(* IEC 61131-3 sources: std_i2980_v2.06_cp053/Source/IMM/ieccontrol/PDP1 (part 3) *)

(* ---- ABRecorderPQ.pu ---- *)
(*
@h    ! WARNING !
@h    The Kemro K2 system (including software) only meets category B according to EN 954-1,
@h    thus it is not intended for usage in safety-relevant control applications in the field
@h    of personal safety (e.g. emergency stop).
@h    To implement potentially necessary safety-relevant control tasks, always use additional
@h    external safety devices that are intended for the particular purpose, and meet the necessary
@h    functional safety.
@h    For further information see EN 954-1 (EN ISO 13849-1) and/or the K2-x00 user manual, chapter
@h    "CE conformity, directives and standards".

*)

IMPORT_OVER_LISTFILE
 START_PROCESS_ALGORITHM
, STOP_PROCESS_ALGORITHM
, GET_SYNC_REFTO
, cCompMold
, tyMovementTrigger
, tevMovementState
, tnOperationMode
, KMB_MeasureBlock2
, KMB_Status
, KMB_CurveResult
, KMB_Curve
, KMB_CreateProfileData
, KSYS_Status
, tevMovementStateData
, KMB_ProfileInfo

END_IMPORT

ALGORITHM_BLOCK ABRecorderPQ #DUMMY_EDIT_BLOCK

SYSTEM_VAR
 sv_TriggerIdxRecPQ : UDINT;
 sv_OperationMode : tnOperationMode ;
 sv_bPQChartHoldRun : BOOL (* PQ chart hold / run *);
END_VAR

SYSTEM_OBJECT
 TaskVis : TASK;
 TaskInject : TASK;
 evMovementState : tevMovementState;
END_OBJECT

VAR
 myMovementTrigger : tyMovementTrigger;
 mevStart : tevMovementState;
 mpbPumpDeviceReady : REFTO BOOL;
 abMeasure : KMB_MeasureBlock2;
 mpiTriggerIdx : REFTO UDINT;
END_VAR

FUNCTION fStartInit : BOOL
 #DUMMY_EDIT_BLOCK
#BEGIN_EDIT_BLOCK
(**************************************** WARNING ********************************************
 *** The KEBA Kemro K2 System including software is not intended for safety control tasks! ***
 ***                       For further information see Comment tab!                        ***
 *********************************************************************************************)

fStartInit := FALSE; //suppress warning about unused formal parameter
START_PROCESS_ALGORITHM(paInit);

;#END_EDIT_BLOCK END_FUNCTION

PROCESS_ALGORITHM paInit ON TaskVis

VAR
 status : KMB_Status;
 curveStatus : KMB_CurveResult;
 curve : KMB_Curve;
 bCreated : BOOL;
 profileData : KMB_CreateProfileData := (ProfileName:='ChartPQ',Type:=KMB_ProfileKind_PDSC,ElementCount:=10000,DataPath:='/protocol/datalogger/',CfgPath:='/workspace/data/ms_config/',ThreadPriority:=6);
 s : KSYS_Status;
END_VAR
#BEGIN_EDIT_BLOCK
(**************************************** WARNING ********************************************
 *** The KEBA Kemro K2 System including software is not intended for safety control tasks! ***
 ***                       For further information see Comment tab!                        ***
 *********************************************************************************************)

// create and init profile 'ChartPQ' of type Mic / 10000  elements
IF (NOT bCreated) THEN
   // create and configure profile for 4 ms cyclic measure
   status := abMeasure.CreateProfile(profileData);
   status := abMeasure.DisableProfileFlashPersistence();
   status := abMeasure.DisableAutoSaveConfig();
   status := abMeasure.SetMeasureTime(T#4ms);
   bCreated := TRUE;
END_IF;

(* add variables 0 .. 3: movement states *)
curve.VariableY := "Mold1.sv_bCloseActive";
curveStatus := abMeasure.AddCurve(curve);

IF (curveStatus.Status = KMB_Status_Not_Connected) THEN
   // see iec library doc and CR_0053873 "KMB_MeasureBlock2: curve is added twice"
   // if a profile has been created it will be installed async. to the IEC task
   // so it may happen that installation of profile has not been finished.
   // we have to repeat here until Status different to "not connected"
   RETURN;
END_IF;

curve.VariableY := "Mold1.sv_bOpenActive";
curveStatus := abMeasure.AddCurve(curve);

curve.VariableY := "Injection1.sv_bPlastActive";
curveStatus := abMeasure.AddCurve(curve);

curve.VariableY := "Injection1.sv_bInjectionActive";
curveStatus := abMeasure.AddCurve(curve);

(* add variables 4 .. 7: PQ set / act master *)
curve.VariableY := "Pump1.sv_KHW_ServoMaster_setValue.rVeloc";
curveStatus := abMeasure.AddCurve(curve);

curve.VariableY := "Pump1.sv_KHW_ServoMaster_actValue.rVeloc";
curveStatus := abMeasure.AddCurve(curve);

curve.VariableY := "Pump1.sv_KHW_ServoMaster_setValue.rAux[1]";
curveStatus := abMeasure.AddCurve(curve);

curve.VariableY := "Pump1.sv_KHW_ServoMaster_actValue.rAux[1]";
curveStatus := abMeasure.AddCurve(curve);

(* add optional variable 8: Q set slave 1 *)
curve.VariableY := "Pump1.sv_KHW_ServoSlave1_actValue.rVeloc";
curveStatus := abMeasure.AddCurve(curve);

(* add optional variable 9: Q set slave 2 *)
curve.VariableY := "Pump1.sv_KHW_ServoSlave2_actValue.rVeloc";
curveStatus := abMeasure.AddCurve(curve);

//////////////////////////////////////////////////////////

// init trigger variables
mpbPumpDeviceReady := GET_SYNC_REFTO("Pump1.sv_bDeviceReady", t#0s, s);
mpiTriggerIdx := @sv_TriggerIdxRecPQ;

//desciption of device and movement id

// mold fwd
myMovementTrigger[1].DeviceId.CompId := cCompMold;
myMovementTrigger[1].DeviceId.IndexId := 1;
myMovementTrigger[1].MoveId := cMoveFwd;
myMovementTrigger[1].MoveDir := cMoveFwd;

// mold bwd
myMovementTrigger[2].DeviceId.CompId := cCompMold;
myMovementTrigger[2].DeviceId.IndexId := 1;
myMovementTrigger[2].MoveId := cMoveBwd;
myMovementTrigger[2].MoveDir := cMoveBwd;

// Inject
myMovementTrigger[3].DeviceId.CompId := cCompInjection;
myMovementTrigger[3].DeviceId.IndexId := 1;
myMovementTrigger[3].MoveId := cMoveInject;
myMovementTrigger[3].MoveDir := cMoveFwd;

// Plast
myMovementTrigger[4].DeviceId.CompId := cCompInjection;
myMovementTrigger[4].DeviceId.IndexId := 1;
myMovementTrigger[4].MoveId := cMovePlast;
myMovementTrigger[4].MoveDir := cMoveBwd;

STOP_PROCESS_ALGORITHM();

;#END_EDIT_BLOCK END_ALGORITHM

EVENT_ALGORITHM evaMovementStart ON TaskInject WITH mevStart

VAR_INPUT
 evMovementStateData : tevMovementStateData;
END_VAR

VAR
 status : KMB_Status;
END_VAR
#BEGIN_EDIT_BLOCK
(**************************************** WARNING ********************************************
 *** The KEBA Kemro K2 System including software is not intended for safety control tasks! ***
 ***                       For further information see Comment tab!                        ***
 *********************************************************************************************)

//Check if in full/half automatic mode
IF sv_OperationMode < nHalfAutomatic THEN
    RETURN;
END_IF;

//Check the movement with the selection on the HMI and the Hold/Run state
//1).Mold close
//2).Mold open
//3).Inject
//4).Plast
IF (evMovementStateData.State = nActive) AND
    ((evMovementStateData.DeviceId = myMovementTrigger[sv_TriggerIdxRecPQ].DeviceId            //movement 1)-> 4)
    AND evMovementStateData.MoveId = myMovementTrigger[sv_TriggerIdxRecPQ].MoveId
    AND evMovementStateData.MoveDir = myMovementTrigger[sv_TriggerIdxRecPQ].MoveDir) OR        //mold close interposition
    (sv_TriggerIdxRecPQ = 1 AND evMovementStateData.DeviceId.CompId = cCompMold AND
     evMovementStateData.DeviceId.IndexId =1 AND evMovementStateData.MoveId = cMoveFwdInterPos AND
     evMovementStateData.MoveDir = cMoveFwd) OR                                           //mold open interposition
    (sv_TriggerIdxRecPQ = 2 AND evMovementStateData.DeviceId.CompId = cCompMold AND
     evMovementStateData.DeviceId.IndexId =1 AND evMovementStateData.MoveId = cMoveBwdInterPos AND
     evMovementStateData.MoveDir = cMoveBwd)) AND (NOT sv_bPQChartHoldRun) THEN

    // start measure
    status := abMeasure.StartMeasure(0);
END_IF;

;#END_EDIT_BLOCK END_ALGORITHM

POSTUPDATE_ALGORITHM pActivateAutoMode ON TaskVis WITH mpiTriggerIdx^

VAR
 status : KMB_Status;
END_VAR
#BEGIN_EDIT_BLOCK
(**************************************** WARNING ********************************************
 *** The KEBA Kemro K2 System including software is not intended for safety control tasks! ***
 ***                       For further information see Comment tab!                        ***
 *********************************************************************************************)

//check if trigger is selected
IF (sv_TriggerIdxRecPQ = 0) THEN
    mevStart := EMPTY;
ELSE
    status := abMeasure.StopMeasure();
    mevStart := evMovementState;
END_IF;

;#END_EDIT_BLOCK END_ALGORITHM

POSTUPDATE_ALGORITHM pActivateManualMode ON TaskInject WITH mpbPumpDeviceReady^

VAR
 status : KMB_Status;
 profileInfo : KMB_ProfileInfo;
END_VAR
#BEGIN_EDIT_BLOCK
(**************************************** WARNING ********************************************
 *** The KEBA Kemro K2 System including software is not intended for safety control tasks! ***
 ***                       For further information see Comment tab!                        ***
 *********************************************************************************************)

// trigger for manual/setup mode ... any movement
IF (sv_OperationMode <= nManual) THEN
    //Check the pump output and Hold/Run function
    IF (NOT mpbPumpDeviceReady^) AND (NOT sv_bPQChartHoldRun)THEN
         profileInfo := abMeasure.GetProfileInfo();
         // if measure still active just keep running ...
         IF (profileInfo.MeasureState = KMB_MeasureState_Inactive) THEN
            status := abMeasure.StartMeasure(0);
         END_IF;
    END_IF;
END_IF;

;#END_EDIT_BLOCK END_ALGORITHM

END_ALGORITHM_BLOCK

#END_OF_IEC_PART

@Puma @IecEditor 6 131 @Pou 25
@@@BEG_Comment@@@
@h    ! WARNING !
@h    The Kemro K2 system (including software) only meets category B according to EN 954-1,
@h    thus it is not intended for usage in safety-relevant control applications in the field
@h    of personal safety (e.g. emergency stop).
@h    To implement potentially necessary safety-relevant control tasks, always use additional
@h    external safety devices that are intended for the particular purpose, and meet the necessary
@h    functional safety.
@h    For further information see EN 954-1 (EN ISO 13849-1) and/or the K2-x00 user manual, chapter
@h    "CE conformity, directives and standards".

@@@END_Comment@@@

@BEG_Contents

@BEG_Func
@RT(17)FuncTreeContainer
3
@Var @RT(23)START_PROCESS_ALGORITHM @RT(0) @T @T @DERIVED 0 @F @RT(23)KEBA_STANDARD_PROCEDURE @F
@T
@BEG_Attrib
0 @RT(0) @RT(0)
@END_Attrib
1 1 @F @F @F @F

@Var @RT(22)STOP_PROCESS_ALGORITHM @RT(0) @T @T @DERIVED 0 @F @RT(23)KEBA_STANDARD_PROCEDURE @F
@T
@BEG_Attrib
0 @RT(0) @RT(0)
@END_Attrib
1 1 @F @F @F @F

@Var @RT(14)GET_SYNC_REFTO @RT(0) @T @T @DERIVED 0 @F @RT(22)KEBA_STANDARD_FUNCTION @F
@T
@BEG_Attrib
0 @RT(0) @RT(0)
@END_Attrib
1 1 @F @F @F @F

@END_Func

@BEG_Const
@RT(18)ConstTreeContainer
1
@Var @RT(9)cCompMold @RT(0) @T @F @DT @RT(4)DINT @RT(0) @T @T @BASIC 0 @F
@F @F
@T
@BEG_Attrib
0 @RT(3)101 @RT(14)Component Mold
@END_Attrib
1 1 @F @F @F @F

@END_Const

@BEG_Export

@BEG_Kind
@ALGORITHM_BLOCK @RT(12)ABRecorderPQ @STRUCTURED_TEXT
@RT(0) @RT(0) @RT(0)
@END_Kind

@BEG_Dcl
@RT(16)DclTreeContainer
11
@Var @RT(7)TaskVis @RT(0) @T @T @RENAMED 0 @T @T @DT @RT(4)TASK @RT(0) @T @T @BASIC 0 @F
@F @F
@T
@BEG_Attrib
3 @RT(0) @RT(0) @RT(0)
@END_Attrib
1 7 @F @F @F @F

@Var @RT(10)TaskInject @RT(0) @T @T @RENAMED 0 @T @T @DT @RT(4)TASK @RT(0) @T @T @BASIC 0 @F
@F @F
@T
@BEG_Attrib
3 @RT(0) @RT(0) @RT(0)
@END_Attrib
1 7 @F @F @F @F

@Var @RT(17)myMovementTrigger @RT(0) @T @T @DERIVED 0 @T @T @DT @RT(17)tyMovementTrigger @RT(0) @T @T @UNKNOWN 0 @F
@F @F
@T
@BEG_Attrib
3 @RT(0) @RT(0) @RT(0)
@END_Attrib
1 0 @F @F @F @F

@Var @RT(15)evMovementState @RT(0) @T @T @DERIVED 0 @T @T @DT @RT(16)tevMovementState @RT(0) @T @T @UNKNOWN 0 @F
@F @F
@T
@BEG_Attrib
3 @RT(0) @RT(0) @RT(0)
@END_Attrib
1 7 @F @F @F @F

@Var @RT(18)sv_TriggerIdxRecPQ @RT(0) @T @F @DT @RT(5)UDINT @RT(0) @T @T @BASIC 0 @F
@F @F
@T
@BEG_Attrib
3 @RT(0) @RT(0) @RT(0)
@END_Attrib
1 8 @F @F @F @F

@Var @RT(16)sv_OperationMode @RT(0) @T @T @DERIVED 0 @T @T @DT @RT(16)tnOperationMode  @RT(0) @T @T @UNKNOWN 0 @F
@F @F
@T
@BEG_Attrib
3 @RT(0) @RT(0) @RT(0)
@END_Attrib
1 8 @F @F @F @F

@Var @RT(18)sv_bPQChartHoldRun @RT(0) @T @F @DT @RT(4)BOOL @RT(0) @T @T @BASIC 0 @F
@F @F
@T
@BEG_Attrib
3 @RT(0) @RT(19)PQ chart hold / run @RT(0)
@END_Attrib
1 8 @F @F @F @F

@Var @RT(8)mevStart @RT(0) @T @T @DERIVED 0 @T @T @DT @RT(16)tevMovementState @RT(0) @T @T @UNKNOWN 0 @F
@F @F
@T
@BEG_Attrib
3 @RT(0) @RT(0) @RT(0)
@END_Attrib
1 0 @F @F @F @F

@Var @RT(18)mpbPumpDeviceReady @RT(0) @T @T @REFTO 0 @T @DT @RT(4)BOOL @RT(0) @T @T @BASIC 0 @F
@F @F
@T
@BEG_Attrib
3 @RT(0) @RT(0) @RT(0)
@END_Attrib
1 0 @F @F @F @F

@Var @RT(9)abMeasure @RT(0) @T @T @DERIVED 0 @T @T @DT @RT(17)KMB_MeasureBlock2 @RT(0) @T @T @UNKNOWN 0 @F
@F @F
@T
@BEG_Attrib
3 @RT(0) @RT(0) @RT(0)
@END_Attrib
1 0 @F @F @F @F

@Var @RT(13)mpiTriggerIdx @RT(0) @T @T @REFTO 0 @T @DT @RT(5)UDINT @RT(0) @T @T @BASIC 0 @F
@F @F
@T
@BEG_Attrib
3 @RT(0) @RT(0) @RT(0)
@END_Attrib
1 0 @F @F @F @F

@END_Dcl

@END_Export

@BEG_Body

5

@BEG_Export

@BEG_Algo
@FUNCTION @RT(10)fStartInit @STRUCTURED_TEXT
@RT(4)BOOL @RT(0) @RT(0) @F @F
@END_Algo

@BEG_Dcl
@RT(16)DclTreeContainer
0
@END_Dcl

@END_Export

@BEG_Export

@BEG_Algo
@PROCESS_ALGORITHM @RT(6)paInit @STRUCTURED_TEXT
@RT(0) @RT(0) @RT(7)TaskVis @F @F
@END_Algo

@BEG_Dcl
@RT(16)DclTreeContainer
6
@Var @RT(6)status @RT(0) @T @T @DERIVED 0 @T @T @DT @RT(10)KMB_Status @RT(0) @T @T @UNKNOWN 0 @F
@F @F
@T
@BEG_Attrib
3 @RT(0) @RT(0) @RT(0)
@END_Attrib
1 0 @F @F @F @F

@Var @RT(11)curveStatus @RT(0) @T @T @DERIVED 0 @T @T @DT @RT(15)KMB_CurveResult @RT(0) @T @T @UNKNOWN 0 @F
@F @F
@T
@BEG_Attrib
3 @RT(0) @RT(0) @RT(0)
@END_Attrib
1 0 @F @F @F @F

@Var @RT(5)curve @RT(0) @T @T @DERIVED 0 @T @T @DT @RT(9)KMB_Curve @RT(0) @T @T @UNKNOWN 0 @F
@F @F
@T
@BEG_Attrib
3 @RT(0) @RT(0) @RT(0)
@END_Attrib
1 0 @F @F @F @F

@Var @RT(8)bCreated @RT(0) @T @T @RENAMED 0 @T @T @DT @RT(4)BOOL @RT(0) @T @T @BASIC 0 @F
@F @F
@T
@BEG_Attrib
3 @RT(0) @RT(0) @RT(0)
@END_Attrib
1 0 @F @F @F @F

@Var @RT(11)profileData @RT(0) @T @T @DERIVED 0 @T @T @DT @RT(21)KMB_CreateProfileData @RT(0) @T @T @UNKNOWN 0 @F
@F @F
@T
@BEG_Attrib
3 @RT(161)(ProfileName:='ChartPQ',Type:=KMB_ProfileKind_PDSC,ElementCount:=10000,DataPath:='/protocol/datalogger/',CfgPath:='/workspace/data/ms_config/',ThreadPriority:=6) @RT(0) @RT(0)
@END_Attrib
1 0 @F @F @F @F

@Var @RT(1)s @RT(0) @T @T @DERIVED 0 @T @T @DT @RT(11)KSYS_Status @RT(0) @T @T @UNKNOWN 0 @F
@F @F
@T
@BEG_Attrib
3 @RT(0) @RT(0) @RT(0)
@END_Attrib
1 0 @F @F @F @F

@END_Dcl

@END_Export

@BEG_Export

@BEG_Algo
@EVENT_ALGORITHM @RT(16)evaMovementStart @STRUCTURED_TEXT
@RT(0) @RT(8)mevStart @RT(10)TaskInject @F @F
@END_Algo

@BEG_Dcl
@RT(16)DclTreeContainer
2
@Var @RT(19)evMovementStateData @RT(0) @T @T @DERIVED 0 @T @T @DT @RT(20)tevMovementStateData @RT(0) @T @T @UNKNOWN 0 @F
@F @F
@T
@BEG_Attrib
3 @RT(0) @RT(0) @RT(0)
@END_Attrib
1 1 @F @F @F @F

@Var @RT(6)status @RT(0) @T @T @DERIVED 0 @T @T @DT @RT(10)KMB_Status @RT(0) @T @T @UNKNOWN 0 @F
@F @F
@T
@BEG_Attrib
3 @RT(0) @RT(0) @RT(0)
@END_Attrib
1 0 @F @F @F @F

@END_Dcl

@END_Export

@BEG_Export

@BEG_Algo
@POSTUPDATE_ALGORITHM @RT(17)pActivateAutoMode @STRUCTURED_TEXT
@RT(0) @RT(14)mpiTriggerIdx^ @RT(7)TaskVis @F @F
@END_Algo

@BEG_Dcl
@RT(16)DclTreeContainer
1
@Var @RT(6)status @RT(0) @T @T @DERIVED 0 @T @T @DT @RT(10)KMB_Status @RT(0) @T @T @UNKNOWN 0 @F
@F @F
@T
@BEG_Attrib
3 @RT(0) @RT(0) @RT(0)
@END_Attrib
1 0 @F @F @F @F

@END_Dcl

@END_Export

@BEG_Export

@BEG_Algo
@POSTUPDATE_ALGORITHM @RT(19)pActivateManualMode @STRUCTURED_TEXT
@RT(0) @RT(19)mpbPumpDeviceReady^ @RT(10)TaskInject @F @F
@END_Algo

@BEG_Dcl
@RT(16)DclTreeContainer
2
@Var @RT(6)status @RT(0) @T @T @DERIVED 0 @T @T @DT @RT(10)KMB_Status @RT(0) @T @T @UNKNOWN 0 @F
@F @F
@T
@BEG_Attrib
3 @RT(0) @RT(0) @RT(0)
@END_Attrib
1 0 @F @F @F @F

@Var @RT(11)profileInfo @RT(0) @T @T @DERIVED 0 @T @T @DT @RT(15)KMB_ProfileInfo @RT(0) @T @T @UNKNOWN 0 @F
@F @F
@T
@BEG_Attrib
3 @RT(0) @RT(0) @RT(0)
@END_Attrib
1 0 @F @F @F @F

@END_Dcl

@END_Export

@BEG_Body
@TL(8)
(**************************************** WARNING ********************************************
 *** The KEBA Kemro K2 System including software is not intended for safety control tasks! ***
 ***                       For further information see Comment tab!                        ***
 *********************************************************************************************)

fStartInit := FALSE; //suppress warning about unused formal parameter
START_PROCESS_ALGORITHM(paInit);

@END_Body

@@@BEG_Comment@@@
@TL(0)

@@@END_Comment@@@

@BEG_Body
@TL(94)
(**************************************** WARNING ********************************************
 *** The KEBA Kemro K2 System including software is not intended for safety control tasks! ***
 ***                       For further information see Comment tab!                        ***
 *********************************************************************************************)

// create and init profile 'ChartPQ' of type Mic / 10000  elements
IF (NOT bCreated) THEN
   // create and configure profile for 4 ms cyclic measure
   status := abMeasure.CreateProfile(profileData);
   status := abMeasure.DisableProfileFlashPersistence();
   status := abMeasure.DisableAutoSaveConfig();
   status := abMeasure.SetMeasureTime(T#4ms);
   bCreated := TRUE;
END_IF;

(* add variables 0 .. 3: movement states *)
curve.VariableY := "Mold1.sv_bCloseActive";
curveStatus := abMeasure.AddCurve(curve);

IF (curveStatus.Status = KMB_Status_Not_Connected) THEN
   // see iec library doc and CR_0053873 "KMB_MeasureBlock2: curve is added twice"
   // if a profile has been created it will be installed async. to the IEC task
   // so it may happen that installation of profile has not been finished.
   // we have to repeat here until Status different to "not connected"
   RETURN;
END_IF;

curve.VariableY := "Mold1.sv_bOpenActive";
curveStatus := abMeasure.AddCurve(curve);

curve.VariableY := "Injection1.sv_bPlastActive";
curveStatus := abMeasure.AddCurve(curve);

curve.VariableY := "Injection1.sv_bInjectionActive";
curveStatus := abMeasure.AddCurve(curve);

(* add variables 4 .. 7: PQ set / act master *)
curve.VariableY := "Pump1.sv_KHW_ServoMaster_setValue.rVeloc";
curveStatus := abMeasure.AddCurve(curve);

curve.VariableY := "Pump1.sv_KHW_ServoMaster_actValue.rVeloc";
curveStatus := abMeasure.AddCurve(curve);

curve.VariableY := "Pump1.sv_KHW_ServoMaster_setValue.rAux[1]";
curveStatus := abMeasure.AddCurve(curve);

curve.VariableY := "Pump1.sv_KHW_ServoMaster_actValue.rAux[1]";
curveStatus := abMeasure.AddCurve(curve);

(* add optional variable 8: Q set slave 1 *)
curve.VariableY := "Pump1.sv_KHW_ServoSlave1_actValue.rVeloc";
curveStatus := abMeasure.AddCurve(curve);

(* add optional variable 9: Q set slave 2 *)
curve.VariableY := "Pump1.sv_KHW_ServoSlave2_actValue.rVeloc";
curveStatus := abMeasure.AddCurve(curve);

//////////////////////////////////////////////////////////

// init trigger variables
mpbPumpDeviceReady := GET_SYNC_REFTO("Pump1.sv_bDeviceReady", t#0s, s);
mpiTriggerIdx := @sv_TriggerIdxRecPQ;

//desciption of device and movement id

// mold fwd
myMovementTrigger[1].DeviceId.CompId := cCompMold;
myMovementTrigger[1].DeviceId.IndexId := 1;
myMovementTrigger[1].MoveId := cMoveFwd;
myMovementTrigger[1].MoveDir := cMoveFwd;

// mold bwd
myMovementTrigger[2].DeviceId.CompId := cCompMold;
myMovementTrigger[2].DeviceId.IndexId := 1;
myMovementTrigger[2].MoveId := cMoveBwd;
myMovementTrigger[2].MoveDir := cMoveBwd;

// Inject
myMovementTrigger[3].DeviceId.CompId := cCompInjection;
myMovementTrigger[3].DeviceId.IndexId := 1;
myMovementTrigger[3].MoveId := cMoveInject;
myMovementTrigger[3].MoveDir := cMoveFwd;

// Plast
myMovementTrigger[4].DeviceId.CompId := cCompInjection;
myMovementTrigger[4].DeviceId.IndexId := 1;
myMovementTrigger[4].MoveId := cMovePlast;
myMovementTrigger[4].MoveDir := cMoveBwd;

STOP_PROCESS_ALGORITHM();

@END_Body

@@@BEG_Comment@@@
@TL(0)

@@@END_Comment@@@

@BEG_Body
@TL(30)
(**************************************** WARNING ********************************************
 *** The KEBA Kemro K2 System including software is not intended for safety control tasks! ***
 ***                       For further information see Comment tab!                        ***
 *********************************************************************************************)

//Check if in full/half automatic mode
IF sv_OperationMode < nHalfAutomatic THEN
    RETURN;
END_IF;

//Check the movement with the selection on the HMI and the Hold/Run state
//1).Mold close
//2).Mold open
//3).Inject
//4).Plast
IF (evMovementStateData.State = nActive) AND
    ((evMovementStateData.DeviceId = myMovementTrigger[sv_TriggerIdxRecPQ].DeviceId            //movement 1)-> 4)
    AND evMovementStateData.MoveId = myMovementTrigger[sv_TriggerIdxRecPQ].MoveId
    AND evMovementStateData.MoveDir = myMovementTrigger[sv_TriggerIdxRecPQ].MoveDir) OR        //mold close interposition
    (sv_TriggerIdxRecPQ = 1 AND evMovementStateData.DeviceId.CompId = cCompMold AND
     evMovementStateData.DeviceId.IndexId =1 AND evMovementStateData.MoveId = cMoveFwdInterPos AND
     evMovementStateData.MoveDir = cMoveFwd) OR                                           //mold open interposition
    (sv_TriggerIdxRecPQ = 2 AND evMovementStateData.DeviceId.CompId = cCompMold AND
     evMovementStateData.DeviceId.IndexId =1 AND evMovementStateData.MoveId = cMoveBwdInterPos AND
     evMovementStateData.MoveDir = cMoveBwd)) AND (NOT sv_bPQChartHoldRun) THEN

    // start measure
    status := abMeasure.StartMeasure(0);
END_IF;

@END_Body

@@@BEG_Comment@@@
@TL(0)

@@@END_Comment@@@

@BEG_Body
@TL(13)
(**************************************** WARNING ********************************************
 *** The KEBA Kemro K2 System including software is not intended for safety control tasks! ***
 ***                       For further information see Comment tab!                        ***
 *********************************************************************************************)

//check if trigger is selected
IF (sv_TriggerIdxRecPQ = 0) THEN
    mevStart := EMPTY;
ELSE
    status := abMeasure.StopMeasure();
    mevStart := evMovementState;
END_IF;

@END_Body

@@@BEG_Comment@@@
@TL(0)

@@@END_Comment@@@

@BEG_Body
@TL(17)
(**************************************** WARNING ********************************************
 *** The KEBA Kemro K2 System including software is not intended for safety control tasks! ***
 ***                       For further information see Comment tab!                        ***
 *********************************************************************************************)

// trigger for manual/setup mode ... any movement
IF (sv_OperationMode <= nManual) THEN
    //Check the pump output and Hold/Run function
    IF (NOT mpbPumpDeviceReady^) AND (NOT sv_bPQChartHoldRun)THEN
         profileInfo := abMeasure.GetProfileInfo();
         // if measure still active just keep running ...
         IF (profileInfo.MeasureState = KMB_MeasureState_Inactive) THEN
            status := abMeasure.StartMeasure(0);
         END_IF;
    END_IF;
END_IF;

@END_Body

@@@BEG_Comment@@@
@TL(0)

@@@END_Comment@@@
@END_Body

@END_Contents

(* ---- FBPDProfileMap.pu ---- *)
IMPORT_OVER_LISTFILE
 KCAT_GetNext
, KCAT_GetValue
, tySpcSettingsArray
, tsPdProfileMap
, KCAT_HandleData
, KCAT_TypeData
, KCAT_NameData
, KCAT_Status

END_IMPORT

FUNCTION_BLOCK FBPDProfileMap #DUMMY_EDIT_BLOCK

VAR_INPUT
 sProfileName : STRING(64);
 pProfileSettings : REFTO tySpcSettingsArray;
END_VAR

VAR_OUTPUT
 ProfileMap : tsPdProfileMap;
END_VAR

VAR_TEMP
 I : USINT;
END_VAR

VAR
 CatHandle : KCAT_HandleData;
 CatType : KCAT_TypeData;
 CatVarNode : KCAT_HandleData;
 CatName : KCAT_NameData;
 Status : KCAT_Status;
 ProfileMapEmpty : tsPdProfileMap := (ProfileIndex:=0);
 sCatName : STRING(255);
 sCatVarName : STRING(255);
 sCatValue : STRING(255);
 iPos : INT;
 iVarId : USINT;
 sVarId : STRING(5);
END_VAR
#BEGIN_EDIT_BLOCK
(**************************************** WARNING ********************************************
 *** The KEBA Kemro K2 System including software is not intended for safety control tasks! ***
 ***                       For further information see Comment tab!                        ***
 *********************************************************************************************)

(* This function block calculates the variable mapping between the
 * single event structure from the profile error event and the
 * error reaction array given in pProfileSettings *)

ProfileMap := ProfileMapEmpty;
ProfileMap.ProfileIndex := 0;

IF (sProfileName = '' OR pProfileSettings = EMPTY) THEN
   RETURN;
END_IF;

sCatName := CONCAT('MS.Profile.', sProfileName);
sCatName := CONCAT(sCatName, '.Param');

CatHandle := KCAT_GetHandle(sCatName);
IF CatHandle.Status <> KCAT_Status_OK THEN
   RETURN;
END_IF;

CatHandle := KCAT_GetFirst(CatHandle.Handle);
sCatName := CONCAT(sCatName, '.ProfileIndex');

WHILE(CatHandle.Status = KCAT_Status_OK) DO

   CatName := KCAT_GetName(CatHandle.Handle);
   CatType := KCAT_GetType(CatHandle.Handle);

   IF (CatName.Name = sCatName) THEN
      (* MS.Profile.<name>.Param.ProfileIndex *)
      Status := KCAT_GetValue(CatHandle.Handle, ProfileMap.ProfileIndex);
   ELSIF (CatType.Type = KCAT_Type_None) THEN
     (* MS.Profile.<name>.Param.Var_<id>.VarName *)
      sCatVarName := CONCAT(CatName.Name, '.VarName');
      CatVarNode := KCAT_GetHandle(sCatVarName);
      IF (CatVarNode.Status = KCAT_Status_OK) THEN
         (* Get variable name *)
         Status := KCAT_GetValue(CatVarNode.Handle, sCatValue);
         (* Find variable ID *)
         iPos := FIND(CatName.Name, '.Var_');
         IF (iPos > 0) THEN
            sVarId := RIGHT(CatName.Name, LEN(CatName.Name) - (iPos + 4));
            iVarId := STRING_TO_USINT(sVarId);
            IF (iVarId >= GET_LOW_BOUND(ProfileMap.Map) AND iVarId <= GET_HIGH_BOUND(ProfileMap.Map)) THEN
               FOR I := GET_LOW_BOUND(pProfileSettings^) TO GET_HIGH_BOUND(pProfileSettings^) DO
                  (* Search for variable name in PDP settings *)
                  IF (pProfileSettings^[I].Variable = sCatValue) THEN
                     ProfileMap.Map[iVarId] := I;
                  END_IF;
               END_FOR;
            END_IF;
         END_IF;

      END_IF;
   END_IF;
   CatHandle := KCAT_GetNext(CatHandle.Handle);

END_WHILE;

;#END_EDIT_BLOCK END_FUNCTION_BLOCK

#END_OF_IEC_PART

@Puma @IecEditor 6 145 @Pou 25
@@@BEG_Comment@@@

@@@END_Comment@@@

@BEG_Contents

@BEG_Func
@RT(17)FuncTreeContainer
2
@Var @RT(12)KCAT_GetNext @RT(0) @T @T @DERIVED 0 @F @RT(22)KEBA_STANDARD_FUNCTION @F
@T
@BEG_Attrib
0 @RT(0) @RT(0)
@END_Attrib
1 1 @F @F @F @F

@Var @RT(13)KCAT_GetValue @RT(0) @T @T @DERIVED 0 @F @RT(22)KEBA_STANDARD_FUNCTION @F
@T
@BEG_Attrib
0 @RT(0) @RT(0)
@END_Attrib
1 1 @F @F @F @F

@END_Func

@BEG_Const
@RT(18)ConstTreeContainer
0
@END_Const

@BEG_Export

@BEG_Kind
@FUNCTION_BLOCK @RT(14)FBPDProfileMap @STRUCTURED_TEXT
@RT(0) @RT(0) @RT(0)
@END_Kind

@BEG_Dcl
@RT(16)DclTreeContainer
16
@Var @RT(12)sProfileName @RT(0) @T @F @DT @RT(10)STRING(64) @RT(0) @T @T @STRING 0 @F @RT(2)64 @F
@F @F
@T
@BEG_Attrib
3 @RT(0) @RT(0) @RT(0)
@END_Attrib
1 1 @F @F @F @F

@Var @RT(16)pProfileSettings @RT(0) @T @T @REFTO 0 @F @DERIVED 0 @T @T @DT @RT(18)tySpcSettingsArray @RT(0) @T @T @UNKNOWN 0 @F
@F @F
@T
@BEG_Attrib
3 @RT(0) @RT(0) @RT(0)
@END_Attrib
1 1 @F @F @F @F

@Var @RT(10)ProfileMap @RT(0) @T @T @DERIVED 0 @T @T @DT @RT(14)tsPdProfileMap @RT(0) @T @T @UNKNOWN 0 @F
@F @F
@T
@BEG_Attrib
3 @RT(0) @RT(0) @RT(0)
@END_Attrib
1 3 @F @F @F @F

@Var @RT(9)CatHandle @RT(0) @T @T @DERIVED 0 @T @T @DT @RT(15)KCAT_HandleData @RT(0) @T @T @UNKNOWN 0 @F
@F @F
@T
@BEG_Attrib
3 @RT(0) @RT(0) @RT(0)
@END_Attrib
1 0 @F @F @F @F

@Var @RT(7)CatType @RT(0) @T @T @DERIVED 0 @T @T @DT @RT(13)KCAT_TypeData @RT(0) @T @T @UNKNOWN 0 @F
@F @F
@T
@BEG_Attrib
3 @RT(0) @RT(0) @RT(0)
@END_Attrib
1 0 @F @F @F @F

@Var @RT(10)CatVarNode @RT(0) @T @T @DERIVED 0 @T @T @DT @RT(15)KCAT_HandleData @RT(0) @T @T @UNKNOWN 0 @F
@F @F
@T
@BEG_Attrib
3 @RT(0) @RT(0) @RT(0)
@END_Attrib
1 0 @F @F @F @F

@Var @RT(7)CatName @RT(0) @T @T @DERIVED 0 @T @T @DT @RT(13)KCAT_NameData @RT(0) @T @T @UNKNOWN 0 @F
@F @F
@T
@BEG_Attrib
3 @RT(0) @RT(0) @RT(0)
@END_Attrib
1 0 @F @F @F @F

@Var @RT(6)Status @RT(0) @T @T @DERIVED 0 @T @T @DT @RT(11)KCAT_Status @RT(0) @T @T @UNKNOWN 0 @F
@F @F
@T
@BEG_Attrib
3 @RT(0) @RT(0) @RT(0)
@END_Attrib
1 0 @F @F @F @F

@Var @RT(15)ProfileMapEmpty @RT(0) @T @T @DERIVED 0 @T @T @DT @RT(14)tsPdProfileMap @RT(0) @T @T @UNKNOWN 0 @F
@F @F
@T
@BEG_Attrib
3 @RT(17)(ProfileIndex:=0) @RT(0) @RT(0)
@END_Attrib
1 0 @F @F @F @F

@Var @RT(8)sCatName @RT(0) @T @F @DT @RT(11)STRING(255) @RT(0) @T @T @STRING 0 @F @RT(3)255 @F
@F @F
@T
@BEG_Attrib
3 @RT(0) @RT(0) @RT(0)
@END_Attrib
1 0 @F @F @F @F

@Var @RT(11)sCatVarName @RT(0) @T @F @DT @RT(11)STRING(255) @RT(0) @T @T @STRING 0 @F @RT(3)255 @F
@F @F
@T
@BEG_Attrib
3 @RT(0) @RT(0) @RT(0)
@END_Attrib
1 0 @F @F @F @F

@Var @RT(9)sCatValue @RT(0) @T @F @DT @RT(11)STRING(255) @RT(0) @T @T @STRING 0 @F @RT(3)255 @F
@F @F
@T
@BEG_Attrib
3 @RT(0) @RT(0) @RT(0)
@END_Attrib
1 0 @F @F @F @F

@Var @RT(4)iPos @RT(0) @T @F @DT @RT(3)INT @RT(0) @T @T @BASIC 0 @F
@F @F
@T
@BEG_Attrib
3 @RT(0) @RT(0) @RT(0)
@END_Attrib
1 0 @F @F @F @F

@Var @RT(6)iVarId @RT(0) @T @F @DT @RT(5)USINT @RT(0) @T @T @BASIC 0 @F
@F @F
@T
@BEG_Attrib
3 @RT(0) @RT(0) @RT(0)
@END_Attrib
1 0 @F @F @F @F

@Var @RT(6)sVarId @RT(0) @T @F @DT @RT(9)STRING(5) @RT(0) @T @T @STRING 0 @F @RT(1)5 @F
@F @F
@T
@BEG_Attrib
3 @RT(0) @RT(0) @RT(0)
@END_Attrib
1 0 @F @F @F @F

@Var @RT(1)I @RT(0) @T @F @DT @RT(5)USINT @RT(0) @T @T @BASIC 0 @F
@F @F
@T
@BEG_Attrib
3 @RT(0) @RT(0) @RT(0)
@END_Attrib
1 4 @F @F @F @F

@END_Dcl

@END_Export

@BEG_Body
@TL(63)
(**************************************** WARNING ********************************************
 *** The KEBA Kemro K2 System including software is not intended for safety control tasks! ***
 ***                       For further information see Comment tab!                        ***
 *********************************************************************************************)

(* This function block calculates the variable mapping between the
 * single event structure from the profile error event and the
 * error reaction array given in pProfileSettings *)

ProfileMap := ProfileMapEmpty;
ProfileMap.ProfileIndex := 0;

IF (sProfileName = '' OR pProfileSettings = EMPTY) THEN
   RETURN;
END_IF;

sCatName := CONCAT('MS.Profile.', sProfileName);
sCatName := CONCAT(sCatName, '.Param');

CatHandle := KCAT_GetHandle(sCatName);
IF CatHandle.Status <> KCAT_Status_OK THEN
   RETURN;
END_IF;

CatHandle := KCAT_GetFirst(CatHandle.Handle);
sCatName := CONCAT(sCatName, '.ProfileIndex');

WHILE(CatHandle.Status = KCAT_Status_OK) DO

   CatName := KCAT_GetName(CatHandle.Handle);
   CatType := KCAT_GetType(CatHandle.Handle);

   IF (CatName.Name = sCatName) THEN
      (* MS.Profile.<name>.Param.ProfileIndex *)
      Status := KCAT_GetValue(CatHandle.Handle, ProfileMap.ProfileIndex);
   ELSIF (CatType.Type = KCAT_Type_None) THEN
     (* MS.Profile.<name>.Param.Var_<id>.VarName *)
      sCatVarName := CONCAT(CatName.Name, '.VarName');
      CatVarNode := KCAT_GetHandle(sCatVarName);
      IF (CatVarNode.Status = KCAT_Status_OK) THEN
         (* Get variable name *)
         Status := KCAT_GetValue(CatVarNode.Handle, sCatValue);
         (* Find variable ID *)
         iPos := FIND(CatName.Name, '.Var_');
         IF (iPos > 0) THEN
            sVarId := RIGHT(CatName.Name, LEN(CatName.Name) - (iPos + 4));
            iVarId := STRING_TO_USINT(sVarId);
            IF (iVarId >= GET_LOW_BOUND(ProfileMap.Map) AND iVarId <= GET_HIGH_BOUND(ProfileMap.Map)) THEN
               FOR I := GET_LOW_BOUND(pProfileSettings^) TO GET_HIGH_BOUND(pProfileSettings^) DO
                  (* Search for variable name in PDP settings *)
                  IF (pProfileSettings^[I].Variable = sCatValue) THEN
                     ProfileMap.Map[iVarId] := I;
                  END_IF;
               END_FOR;
            END_IF;
         END_IF;

      END_IF;
   END_IF;
   CatHandle := KCAT_GetNext(CatHandle.Handle);

END_WHILE;

@END_Body

@END_Contents

(* ---- ABPreShotCounter.pu ---- *)
(*
@h    ! WARNING !
@h    The Kemro K2 system (including software) only meets category B according to EN 954-1,
@h    thus it is not intended for usage in safety-relevant control applications in the field
@h    of personal safety (e.g. emergency stop).
@h    To implement potentially necessary safety-relevant control tasks, always use additional
@h    external safety devices that are intended for the particular purpose, and meet the necessary
@h    functional safety.
@h    For further information see EN 954-1 (EN ISO 13849-1) and/or the K2-x00 user manual, chapter
@h    "CE conformity, directives and standards".

AB for pre - shotcounter movement
- register movement for increasing pre shot counter
- increase sv_iPreShotCounter if start event is received (from FBAutocycle SFC)
- if ODC functionunit is available, the preshot counter is increased automatically after
  mold open movement is started
*)

IMPORT_OVER_LISTFILE
 cCompODC
, tsMoveData
, tevStart
, tevStartedStopped
, tsDeviceId
, tnOperationMode
, tevMovementState
, tyNumberOfDevices
, ABMovementRegister
, tevStartData
, tevStartedStoppedData
, tevMovementStateData

END_IMPORT

ALGORITHM_BLOCK ABPreShotCounter #DUMMY_EDIT_BLOCK

SYSTEM_VAR
 sv_bInitStart : BOOL;
 sv_MovePreShotCounter : tsMoveData;
 sv_DeviceId : tsDeviceId;
 sv_iPreShotCounter : DINT (* shot counter for PDS (increased before ejector movement) *);
 sv_OperationMode : tnOperationMode;
 sv_NumberOfDevices : tyNumberOfDevices;
END_VAR

SYSTEM_OBJECT
 PU_Task_7 : TASK;
 EV_Task_3 : TASK;
 evStart : tevStart;
 evStartedStopped : tevStartedStopped;
 evMovementState : tevMovementState;
END_OBJECT

VAR
 mevMovementState : tevMovementState;
 mevStart : tevStart;
END_VAR

POSTUPDATE_ALGORITHM pInitStart ON PU_Task_7 WITH sv_bInitStart

VAR
 abMovePreShotCounterRegister : ABMovementRegister;
END_VAR
#BEGIN_EDIT_BLOCK
(**************************************** WARNING ********************************************
 *** The KEBA Kemro K2 System including software is not intended for safety control tasks! ***
 ***                       For further information see Comment tab!                        ***
 *********************************************************************************************)

//check if ODC - function unit is available
IF sv_NumberOfDevices[cCompODC] = 1 THEN
   //listen to movement state events
   mevMovementState := evMovementState;
ELSE
   //register movement for pre shotcounter increasing
   //this is necessary because autocycle SFC sends a start event for this movement
   abMovePreShotCounterRegister.aRegister(@sv_MovePreShotCounter);

   //listen to start events
   mevStart := evStart;
END_IF;

;#END_EDIT_BLOCK END_ALGORITHM

ALGORITHM aIncrease

#BEGIN_EDIT_BLOCK
(**************************************** WARNING ********************************************
 *** The KEBA Kemro K2 System including software is not intended for safety control tasks! ***
 ***                       For further information see Comment tab!                        ***
 *********************************************************************************************)

//increase pre shot counter
IF sv_OperationMode >= nHalfAutomatic THEN
    sv_iPreShotCounter := sv_iPreShotCounter + 1;
END_IF;

;#END_EDIT_BLOCK END_ALGORITHM

EVENT_ALGORITHM evaStart ON EV_Task_3 WITH mevStart

VAR_INPUT
 evStartData : tevStartData;
END_VAR

VAR
 evStartedStoppedData : tevStartedStoppedData;
END_VAR
#BEGIN_EDIT_BLOCK
(**************************************** WARNING ********************************************
 *** The KEBA Kemro K2 System including software is not intended for safety control tasks! ***
 ***                       For further information see Comment tab!                        ***
 *********************************************************************************************)

IF evStartData.DeviceId <> sv_DeviceId THEN
   RETURN;
END_IF;

IF evStartData.MoveDir = sv_MovePreShotCounter.MoveDir AND evStartData.MoveId = sv_MovePreShotCounter.MoveId THEN
   // The evStartedStopped events are necessary because of the ODC,
   // which keeps a list of running movements.
   // Elements are added before a evStart is sent
   // and removed on evStartedStopped nStopped/nStartNotAllowed.
   // When no evStartedStopped are sent the shotcounter increase movements are never removed again

   // send started-Message
   evStartedStoppedData.DeviceId := sv_DeviceId;
   evStartedStoppedData.MoveId := sv_MovePreShotCounter.MoveId;
   evStartedStoppedData.MoveDir := sv_MovePreShotCounter.MoveDir;
   evStartedStoppedData.State := nStarted;
   SET_EVENT(evStartedStopped,evStartedStoppedData);

   aIncrease();

   // send stopped-Message
   evStartedStoppedData.State := nStopped;
   SET_EVENT(evStartedStopped,evStartedStoppedData);
END_IF;

;#END_EDIT_BLOCK END_ALGORITHM

EVENT_ALGORITHM evaMovementState ON EV_Task_3 WITH mevMovementState

VAR_INPUT
 evMovementStateData : tevMovementStateData;
END_VAR

VAR
 DeviceIdMold : tsDeviceId := (CompId:=cCompMold,IndexId:=1);
END_VAR
#BEGIN_EDIT_BLOCK
(**************************************** WARNING ********************************************
 *** The KEBA Kemro K2 System including software is not intended for safety control tasks! ***
 ***                       For further information see Comment tab!                        ***
 *********************************************************************************************)

IF evMovementStateData.State = nInactive THEN
   RETURN;
END_IF;

IF evMovementStateData.DeviceId = DeviceIdMold AND evMovementStateData.MoveId = cMoveBwd THEN
   //mold open started -> increase pre shotcounter
   aIncrease();
END_IF;

;#END_EDIT_BLOCK END_ALGORITHM

END_ALGORITHM_BLOCK

#END_OF_IEC_PART

@Puma @IecEditor 6 97 @Pou 25
@@@BEG_Comment@@@
@h    ! WARNING !
@h    The Kemro K2 system (including software) only meets category B according to EN 954-1,
@h    thus it is not intended for usage in safety-relevant control applications in the field
@h    of personal safety (e.g. emergency stop).
@h    To implement potentially necessary safety-relevant control tasks, always use additional
@h    external safety devices that are intended for the particular purpose, and meet the necessary
@h    functional safety.
@h    For further information see EN 954-1 (EN ISO 13849-1) and/or the K2-x00 user manual, chapter
@h    "CE conformity, directives and standards".

AB for pre - shotcounter movement
- register movement for increasing pre shot counter
- increase sv_iPreShotCounter if start event is received (from FBAutocycle SFC)
- if ODC functionunit is available, the preshot counter is increased automatically after
  mold open movement is started
@@@END_Comment@@@

@BEG_Contents

@BEG_Func
@RT(17)FuncTreeContainer
0
@END_Func

@BEG_Const
@RT(18)ConstTreeContainer
1
@Var @RT(8)cCompODC @RT(0) @T @F @DT @RT(4)DINT @RT(0) @T @T @BASIC 0 @F
@F @F
@T
@BEG_Attrib
0 @RT(3)136 @RT(13)Component ODC
@END_Attrib
1 1 @F @F @F @F

@END_Const

@BEG_Export

@BEG_Kind
@ALGORITHM_BLOCK @RT(16)ABPreShotCounter @STRUCTURED_TEXT
@RT(0) @RT(0) @RT(0)
@END_Kind

@BEG_Dcl
@RT(16)DclTreeContainer
13
@Var @RT(9)PU_Task_7 @RT(0) @T @F @DT @RT(4)TASK @RT(0) @T @T @BASIC 0 @F
@F @F
@T
@BEG_Attrib
3 @RT(0) @RT(0) @RT(0)
@END_Attrib
1 7 @F @F @F @F

@Var @RT(9)EV_Task_3 @RT(0) @T @F @DT @RT(4)TASK @RT(0) @T @T @BASIC 0 @F
@F @F
@T
@BEG_Attrib
3 @RT(0) @RT(0) @RT(0)
@END_Attrib
1 7 @F @F @F @F

@Var @RT(13)sv_bInitStart @RT(0) @T @F @DT @RT(4)BOOL @RT(0) @T @T @BASIC 0 @F
@F @F
@T
@BEG_Attrib
3 @RT(0) @RT(0) @RT(0)
@END_Attrib
1 8 @F @F @F @F

@Var @RT(21)sv_MovePreShotCounter @RT(0) @T @T @DERIVED 0 @T @T @DT @RT(10)tsMoveData @RT(0) @T @T @UNKNOWN 0 @F
@F @F
@T
@BEG_Attrib
3 @RT(0) @RT(0) @RT(0)
@END_Attrib
1 8 @F @F @F @F

@Var @RT(7)evStart @RT(0) @T @T @DERIVED 0 @T @T @DT @RT(8)tevStart @RT(0) @T @T @UNKNOWN 0 @F
@F @F
@T
@BEG_Attrib
3 @RT(0) @RT(0) @RT(0)
@END_Attrib
1 7 @F @F @F @F

@Var @RT(16)evStartedStopped @RT(0) @T @T @DERIVED 0 @T @T @DT @RT(17)tevStartedStopped @RT(0) @T @T @UNKNOWN 0 @F
@F @F
@T
@BEG_Attrib
3 @RT(0) @RT(0) @RT(0)
@END_Attrib
1 7 @F @F @F @F

@Var @RT(11)sv_DeviceId @RT(0) @T @T @DERIVED 0 @T @T @DT @RT(10)tsDeviceId @RT(0) @T @T @UNKNOWN 0 @F
@F @F
@T
@BEG_Attrib
3 @RT(0) @RT(0) @RT(0)
@END_Attrib
1 8 @F @F @F @F

@Var @RT(18)sv_iPreShotCounter @RT(0) @T @F @DT @RT(4)DINT @RT(0) @T @T @BASIC 0 @F
@F @F
@T
@BEG_Attrib
3 @RT(0) @RT(56)shot counter for PDS (increased before ejector movement) @RT(0)
@END_Attrib
1 8 @F @F @F @F

@Var @RT(16)sv_OperationMode @RT(0) @T @T @DERIVED 0 @T @T @DT @RT(15)tnOperationMode @RT(0) @T @T @UNKNOWN 0 @F
@F @F
@T
@BEG_Attrib
3 @RT(0) @RT(0) @RT(0)
@END_Attrib
1 8 @F @F @F @F

@Var @RT(16)mevMovementState @RT(0) @T @T @RENAMED 0 @T @T @DT @RT(16)tevMovementState @RT(0) @T @T @UNKNOWN 0 @F
@F @F
@T
@BEG_Attrib
3 @RT(0) @RT(0) @RT(0)
@END_Attrib
1 0 @F @F @F @F

@Var @RT(18)sv_NumberOfDevices @RT(0) @T @T @DERIVED 0 @T @T @DT @RT(17)tyNumberOfDevices @RT(0) @T @T @UNKNOWN 0 @F
@F @F
@T
@BEG_Attrib
3 @RT(0) @RT(0) @RT(0)
@END_Attrib
1 8 @F @F @F @F

@Var @RT(15)evMovementState @RT(0) @T @T @DERIVED 0 @T @T @DT @RT(16)tevMovementState @RT(0) @T @T @UNKNOWN 0 @F
@F @F
@T
@BEG_Attrib
3 @RT(0) @RT(0) @RT(0)
@END_Attrib
1 7 @F @F @F @F

@Var @RT(8)mevStart @RT(0) @T @T @RENAMED 0 @T @T @DT @RT(8)tevStart @RT(0) @T @T @UNKNOWN 0 @F
@F @F
@T
@BEG_Attrib
3 @RT(0) @RT(0) @RT(0)
@END_Attrib
1 0 @F @F @F @F

@END_Dcl

@END_Export

@BEG_Body

4

@BEG_Export

@BEG_Algo
@POSTUPDATE_ALGORITHM @RT(10)pInitStart @STRUCTURED_TEXT
@RT(0) @RT(13)sv_bInitStart @RT(9)PU_Task_7 @F @F
@END_Algo

@BEG_Dcl
@RT(16)DclTreeContainer
1
@Var @RT(28)abMovePreShotCounterRegister @RT(0) @T @T @DERIVED 0 @T @T @DT @RT(18)ABMovementRegister @RT(0) @T @T @UNKNOWN 0 @F
@F @F
@T
@BEG_Attrib
3 @RT(0) @RT(0) @RT(0)
@END_Attrib
1 0 @F @F @F @F

@END_Dcl

@END_Export

@BEG_Export

@BEG_Algo
@ALGORITHM @RT(9)aIncrease @STRUCTURED_TEXT
@RT(0) @RT(0) @RT(0) @F @F
@END_Algo

@BEG_Dcl
@RT(16)DclTreeContainer
0
@END_Dcl

@END_Export

@BEG_Export

@BEG_Algo
@EVENT_ALGORITHM @RT(8)evaStart @STRUCTURED_TEXT
@RT(0) @RT(8)mevStart @RT(9)EV_Task_3 @F @F
@END_Algo

@BEG_Dcl
@RT(16)DclTreeContainer
2
@Var @RT(11)evStartData @RT(0) @T @T @DERIVED 0 @T @T @DT @RT(12)tevStartData @RT(0) @T @T @UNKNOWN 0 @F
@F @F
@T
@BEG_Attrib
3 @RT(0) @RT(0) @RT(0)
@END_Attrib
1 1 @F @F @F @F

@Var @RT(20)evStartedStoppedData @RT(0) @T @T @DERIVED 0 @T @T @DT @RT(21)tevStartedStoppedData @RT(0) @T @T @UNKNOWN 0 @F
@F @F
@T
@BEG_Attrib
3 @RT(0) @RT(0) @RT(0)
@END_Attrib
1 0 @F @F @F @F

@END_Dcl

@END_Export

@BEG_Export

@BEG_Algo
@EVENT_ALGORITHM @RT(16)evaMovementState @STRUCTURED_TEXT
@RT(0) @RT(16)mevMovementState @RT(9)EV_Task_3 @F @F
@END_Algo

@BEG_Dcl
@RT(16)DclTreeContainer
2
@Var @RT(19)evMovementStateData @RT(0) @T @T @DERIVED 0 @T @T @DT @RT(20)tevMovementStateData @RT(0) @T @T @UNKNOWN 0 @F
@F @F
@T
@BEG_Attrib
3 @RT(0) @RT(0) @RT(0)
@END_Attrib
1 1 @F @F @F @F

@Var @RT(12)DeviceIdMold @RT(0) @T @T @DERIVED 0 @T @T @DT @RT(10)tsDeviceId @RT(0) @T @T @UNKNOWN 0 @F
@F @F
@T
@BEG_Attrib
3 @RT(30)(CompId:=cCompMold,IndexId:=1) @RT(0) @RT(0)
@END_Attrib
1 0 @F @F @F @F

@END_Dcl

@END_Export

@BEG_Body
@TL(18)
(**************************************** WARNING ********************************************
 *** The KEBA Kemro K2 System including software is not intended for safety control tasks! ***
 ***                       For further information see Comment tab!                        ***
 *********************************************************************************************)

//check if ODC - function unit is available
IF sv_NumberOfDevices[cCompODC] = 1 THEN
   //listen to movement state events
   mevMovementState := evMovementState;
ELSE
   //register movement for pre shotcounter increasing
   //this is necessary because autocycle SFC sends a start event for this movement
   abMovePreShotCounterRegister.aRegister(@sv_MovePreShotCounter);

   //listen to start events
   mevStart := evStart;
END_IF;

@END_Body

@@@BEG_Comment@@@
@TL(0)

@@@END_Comment@@@

@BEG_Body
@TL(10)
(**************************************** WARNING ********************************************
 *** The KEBA Kemro K2 System including software is not intended for safety control tasks! ***
 ***                       For further information see Comment tab!                        ***
 *********************************************************************************************)

//increase pre shot counter
IF sv_OperationMode >= nHalfAutomatic THEN
    sv_iPreShotCounter := sv_iPreShotCounter + 1;
END_IF;

@END_Body

@@@BEG_Comment@@@
@TL(0)

@@@END_Comment@@@

@BEG_Body
@TL(30)
(**************************************** WARNING ********************************************
 *** The KEBA Kemro K2 System including software is not intended for safety control tasks! ***
 ***                       For further information see Comment tab!                        ***
 *********************************************************************************************)

IF evStartData.DeviceId <> sv_DeviceId THEN
   RETURN;
END_IF;

IF evStartData.MoveDir = sv_MovePreShotCounter.MoveDir AND evStartData.MoveId = sv_MovePreShotCounter.MoveId THEN
   // The evStartedStopped events are necessary because of the ODC,
   // which keeps a list of running movements.
   // Elements are added before a evStart is sent
   // and removed on evStartedStopped nStopped/nStartNotAllowed.
   // When no evStartedStopped are sent the shotcounter increase movements are never removed again

   // send started-Message
   evStartedStoppedData.DeviceId := sv_DeviceId;
   evStartedStoppedData.MoveId := sv_MovePreShotCounter.MoveId;
   evStartedStoppedData.MoveDir := sv_MovePreShotCounter.MoveDir;
   evStartedStoppedData.State := nStarted;
   SET_EVENT(evStartedStopped,evStartedStoppedData);

   aIncrease();

   // send stopped-Message
   evStartedStoppedData.State := nStopped;
   SET_EVENT(evStartedStopped,evStartedStoppedData);
END_IF;

@END_Body

@@@BEG_Comment@@@
@TL(0)

@@@END_Comment@@@

@BEG_Body
@TL(14)
(**************************************** WARNING ********************************************
 *** The KEBA Kemro K2 System including software is not intended for safety control tasks! ***
 ***                       For further information see Comment tab!                        ***
 *********************************************************************************************)

IF evMovementStateData.State = nInactive THEN
   RETURN;
END_IF;

IF evMovementStateData.DeviceId = DeviceIdMold AND evMovementStateData.MoveId = cMoveBwd THEN
   //mold open started -> increase pre shotcounter
   aIncrease();
END_IF;

@END_Body

@@@BEG_Comment@@@
@TL(0)

@@@END_Comment@@@
@END_Body

@END_Contents

(* ---- ABRecorderCharts.pu ---- *)
(*
@h    ! WARNING !
@h    The Kemro K2 system (including software) only meets category B according to EN 954-1,
@h    thus it is not intended for usage in safety-relevant control applications in the field
@h    of personal safety (e.g. emergency stop).
@h    To implement potentially necessary safety-relevant control tasks, always use additional
@h    external safety devices that are intended for the particular purpose, and meet the necessary
@h    functional safety.
@h    For further information see EN 954-1 (EN ISO 13849-1) and/or the K2-x00 user manual, chapter
@h    "CE conformity, directives and standards".

*)

IMPORT_OVER_LISTFILE
 GET_SYNC_REFTO
, cSubOpSpeedpumpMaster
, cCompEnergyMeter
, ABRecorderPQ
, ABRecorderDriveTemp
, ABRecorderEnergyShot
, ABRecorderEnergyCycle
, KSYS_Status
, tCompId

END_IMPORT

ALGORITHM_BLOCK ABRecorderCharts #DUMMY_EDIT_BLOCK

SYSTEM_OBJECT
 TaskMid : TASK;
END_OBJECT

VAR
 abRecorderPQ : ABRecorderPQ;
 abRecorderDriveTemp : ABRecorderDriveTemp;
 abRecorderEnergyShot : ABRecorderEnergyShot;
 abRecorderEnergyCycle : ABRecorderEnergyCycle;
END_VAR

PROCESS_ALGORITHM paInit ON TaskMid AUTOSTART

VAR
 pOption : REFTO DWORD;
 b : BOOL;
 bIsSpeedPump : BOOL;
 s : KSYS_Status;
 pIsKvb : REFTO DINT;
 pEnergyMeterCompId : REFTO tCompId;
 bHasEnergyMeter : BOOL;
 pUsedServoDrives : REFTO DWORD;
 bHasServoDrives : BOOL;
END_VAR
#BEGIN_EDIT_BLOCK
(**************************************** WARNING ********************************************
 *** The KEBA Kemro K2 System including software is not intended for safety control tasks! ***
 ***                       For further information see Comment tab!                        ***
 *********************************************************************************************)

// kvb system? -> don't start recorder
pIsKvb := GET_SYNC_REFTO('KVB.sv_MaskID', T#0s, s);
IF (s = KSYS_Status_OK) THEN
    STOP_PROCESS_ALGORITHM();
    RETURN;
END_IF;

pOption := GET_SYNC_REFTO('Pump1.sv_Options', T#0s, s);

// any speedpump configuration?
bIsSpeedPump := (s = KSYS_Status_OK)
   AND ((pOption^ AND cSubOpSpeedpumpMaster) = cSubOpSpeedpumpMaster);

IF (bIsSpeedPump) THEN
    b := abRecorderPQ.fStartInit();
    b := abRecorderDriveTemp.fStartInit();
END_IF;

// has servo drives?
pUsedServoDrives := GET_SYNC_REFTO('ServoDrives1.sv_ServoDriveCentral.iUsedDrives', T#0s, s);
bHasServoDrives := (s = KSYS_Status_OK);

IF (bHasServoDrives) THEN
    b := abRecorderEnergyCycle.fStartInit();
END_IF;

// has energy meter?
pEnergyMeterCompId := GET_SYNC_REFTO('EnergyMeter1.sv_DeviceId.CompId', T#0s, s);
bHasEnergyMeter := (s = KSYS_Status_OK);

IF (bHasServoDrives OR bHasEnergyMeter) THEN
    b := abRecorderEnergyShot.fStartInit();
END_IF;

STOP_PROCESS_ALGORITHM();

;#END_EDIT_BLOCK END_ALGORITHM

END_ALGORITHM_BLOCK

#END_OF_IEC_PART

@Puma @IecEditor 6 131 @Pou 25
@@@BEG_Comment@@@
@h    ! WARNING !
@h    The Kemro K2 system (including software) only meets category B according to EN 954-1,
@h    thus it is not intended for usage in safety-relevant control applications in the field
@h    of personal safety (e.g. emergency stop).
@h    To implement potentially necessary safety-relevant control tasks, always use additional
@h    external safety devices that are intended for the particular purpose, and meet the necessary
@h    functional safety.
@h    For further information see EN 954-1 (EN ISO 13849-1) and/or the K2-x00 user manual, chapter
@h    "CE conformity, directives and standards".

@@@END_Comment@@@

@BEG_Contents

@BEG_Func
@RT(17)FuncTreeContainer
1
@Var @RT(14)GET_SYNC_REFTO @RT(0) @T @T @DERIVED 0 @F @RT(22)KEBA_STANDARD_FUNCTION @F
@T
@BEG_Attrib
0 @RT(0) @RT(0)
@END_Attrib
1 1 @F @F @F @F

@END_Func

@BEG_Const
@RT(18)ConstTreeContainer
2
@Var @RT(21)cSubOpSpeedpumpMaster @RT(0) @T @F @DT @RT(5)DWORD @RT(0) @T @T @BASIC 0 @F
@F @F
@T
@BEG_Attrib
0 @RT(6)16#100 @RT(17)Speed pump Master
@END_Attrib
1 1 @F @F @F @F

@Var @RT(16)cCompEnergyMeter @RT(0) @T @F @DT @RT(4)DINT @RT(0) @T @T @BASIC 0 @F
@F @F
@T
@BEG_Attrib
0 @RT(3)157 @RT(22)Component Energy meter
@END_Attrib
1 1 @F @F @F @F

@END_Const

@BEG_Export

@BEG_Kind
@ALGORITHM_BLOCK @RT(16)ABRecorderCharts @STRUCTURED_TEXT
@RT(0) @RT(0) @RT(0)
@END_Kind

@BEG_Dcl
@RT(16)DclTreeContainer
5
@Var @RT(7)TaskMid @RT(0) @T @T @RENAMED 0 @T @T @DT @RT(4)TASK @RT(0) @T @T @BASIC 0 @F
@F @F
@T
@BEG_Attrib
3 @RT(0) @RT(0) @RT(0)
@END_Attrib
1 7 @F @F @F @F

@Var @RT(12)abRecorderPQ @RT(0) @T @T @DERIVED 0 @T @T @DT @RT(12)ABRecorderPQ @RT(0) @T @T @UNKNOWN 0 @F
@F @F
@T
@BEG_Attrib
3 @RT(0) @RT(0) @RT(0)
@END_Attrib
1 0 @F @F @F @F

@Var @RT(19)abRecorderDriveTemp @RT(0) @T @T @DERIVED 0 @T @T @DT @RT(19)ABRecorderDriveTemp @RT(0) @T @T @UNKNOWN 0 @F
@F @F
@T
@BEG_Attrib
3 @RT(0) @RT(0) @RT(0)
@END_Attrib
1 0 @F @F @F @F

@Var @RT(20)abRecorderEnergyShot @RT(0) @T @T @DERIVED 0 @T @T @DT @RT(20)ABRecorderEnergyShot @RT(0) @T @T @UNKNOWN 0 @F
@F @F
@T
@BEG_Attrib
3 @RT(0) @RT(0) @RT(0)
@END_Attrib
1 0 @F @F @F @F

@Var @RT(21)abRecorderEnergyCycle @RT(0) @T @T @DERIVED 0 @T @T @DT @RT(21)ABRecorderEnergyCycle @RT(0) @T @T @UNKNOWN 0 @F
@F @F
@T
@BEG_Attrib
3 @RT(0) @RT(0) @RT(0)
@END_Attrib
1 0 @F @F @F @F

@END_Dcl

@END_Export

@BEG_Body

1

@BEG_Export

@BEG_Algo
@PROCESS_ALGORITHM @RT(6)paInit @STRUCTURED_TEXT
@RT(0) @RT(0) @RT(7)TaskMid @T @F
@END_Algo

@BEG_Dcl
@RT(16)DclTreeContainer
9
@Var @RT(7)pOption @RT(0) @T @T @REFTO 0 @T @DT @RT(5)DWORD @RT(0) @T @T @BASIC 0 @F
@F @F
@T
@BEG_Attrib
3 @RT(0) @RT(0) @RT(0)
@END_Attrib
1 0 @F @F @F @F

@Var @RT(1)b @RT(0) @T @F @DT @RT(4)BOOL @RT(0) @T @T @BASIC 0 @F
@F @F
@T
@BEG_Attrib
3 @RT(0) @RT(0) @RT(0)
@END_Attrib
1 0 @F @F @F @F

@Var @RT(12)bIsSpeedPump @RT(0) @T @F @DT @RT(4)BOOL @RT(0) @T @T @BASIC 0 @F
@F @F
@T
@BEG_Attrib
3 @RT(0) @RT(0) @RT(0)
@END_Attrib
1 0 @F @F @F @F

@Var @RT(1)s @RT(0) @T @T @DERIVED 0 @T @T @DT @RT(11)KSYS_Status @RT(0) @T @T @UNKNOWN 0 @F
@F @F
@T
@BEG_Attrib
3 @RT(0) @RT(0) @RT(0)
@END_Attrib
1 0 @F @F @F @F

@Var @RT(6)pIsKvb @RT(0) @T @T @REFTO 0 @T @DT @RT(4)DINT @RT(0) @T @T @BASIC 0 @F
@F @F
@T
@BEG_Attrib
3 @RT(0) @RT(0) @RT(0)
@END_Attrib
1 0 @F @F @F @F

@Var @RT(18)pEnergyMeterCompId @RT(0) @T @T @REFTO 0 @F @DERIVED 0 @T @T @DT @RT(7)tCompId @RT(0) @T @T @UNKNOWN 0 @F
@F @F
@T
@BEG_Attrib
3 @RT(0) @RT(0) @RT(0)
@END_Attrib
1 0 @F @F @F @F

@Var @RT(15)bHasEnergyMeter @RT(0) @T @F @DT @RT(4)BOOL @RT(0) @T @T @BASIC 0 @F
@F @F
@T
@BEG_Attrib
3 @RT(0) @RT(0) @RT(0)
@END_Attrib
1 0 @F @F @F @F

@Var @RT(16)pUsedServoDrives @RT(0) @T @T @REFTO 0 @T @DT @RT(5)DWORD @RT(0) @T @T @BASIC 0 @F
@F @F
@T
@BEG_Attrib
3 @RT(0) @RT(0) @RT(0)
@END_Attrib
1 0 @F @F @F @F

@Var @RT(15)bHasServoDrives @RT(0) @T @F @DT @RT(4)BOOL @RT(0) @T @T @BASIC 0 @F
@F @F
@T
@BEG_Attrib
3 @RT(0) @RT(0) @RT(0)
@END_Attrib
1 0 @F @F @F @F

@END_Dcl

@END_Export

@BEG_Body
@TL(42)
(**************************************** WARNING ********************************************
 *** The KEBA Kemro K2 System including software is not intended for safety control tasks! ***
 ***                       For further information see Comment tab!                        ***
 *********************************************************************************************)

// kvb system? -> don't start recorder
pIsKvb := GET_SYNC_REFTO('KVB.sv_MaskID', T#0s, s);
IF (s = KSYS_Status_OK) THEN
    STOP_PROCESS_ALGORITHM();
    RETURN;
END_IF;

pOption := GET_SYNC_REFTO('Pump1.sv_Options', T#0s, s);

// any speedpump configuration?
bIsSpeedPump := (s = KSYS_Status_OK)
   AND ((pOption^ AND cSubOpSpeedpumpMaster) = cSubOpSpeedpumpMaster);

IF (bIsSpeedPump) THEN
    b := abRecorderPQ.fStartInit();
    b := abRecorderDriveTemp.fStartInit();
END_IF;

// has servo drives?
pUsedServoDrives := GET_SYNC_REFTO('ServoDrives1.sv_ServoDriveCentral.iUsedDrives', T#0s, s);
bHasServoDrives := (s = KSYS_Status_OK);

IF (bHasServoDrives) THEN
    b := abRecorderEnergyCycle.fStartInit();
END_IF;

// has energy meter?
pEnergyMeterCompId := GET_SYNC_REFTO('EnergyMeter1.sv_DeviceId.CompId', T#0s, s);
bHasEnergyMeter := (s = KSYS_Status_OK);

IF (bHasServoDrives OR bHasEnergyMeter) THEN
    b := abRecorderEnergyShot.fStartInit();
END_IF;

STOP_PROCESS_ALGORITHM();

@END_Body

@@@BEG_Comment@@@
@TL(0)

@@@END_Comment@@@
@END_Body

@END_Contents

(* ---- FPlausSPCAction.pu ---- *)
(*
@h    ! WARNING !
@h    The Kemro K2 system (including software) only meets category B according to EN 954-1,
@h    thus it is not intended for usage in safety-relevant control applications in the field
@h    of personal safety (e.g. emergency stop).
@h    To implement potentially necessary safety-relevant control tasks, always use additional
@h    external safety devices that are intended for the particular purpose, and meet the necessary
@h    functional safety.
@h    For further information see EN 954-1 (EN ISO 13849-1) and/or the K2-x00 user manual, chapter
@h    "CE conformity, directives and standards".

Plausibility function for SPC error / warn action
*)

IMPORT_OVER_LISTFILE
 GET_SYNC_REFTO
, cCompEcoRobot
, tsLimitDataINT
, tyNumberOfDevices
, KSYS_Status
, tnRobotInterface

END_IMPORT

PLAUSIBILITY_FUNCTION FPlausSPCAction : tsLimitDataINT

VAR_INPUT
 DeviceClass : INT;
 Userlevel : INT;
END_VAR

SYSTEM_VAR_IN
 sv_NumberOfDevices : tyNumberOfDevices;
END_VAR

VAR
 s : KSYS_Status;
 pbBool : REFTO BOOL;
 pInterfaceType : REFTO tnRobotInterface;
 bScrapModeAllowed : BOOL;
END_VAR
#BEGIN_EDIT_BLOCK
(**************************************** WARNING ********************************************
 *** The KEBA Kemro K2 System including software is not intended for safety control tasks! ***
 ***                       For further information see Comment tab!                        ***
 *********************************************************************************************)

//"hold scrap" mode not allowed if Reject gate is available or
//robot switched on

FPlausSPCAction.iLowerLimit := 0;

bScrapModeAllowed := TRUE;
pbBool := GET_SYNC_REFTO("RejectGate1.do_RejectGate", T#0s, s);
IF s = KSYS_Status_OK THEN
   //reject gate available
   bScrapModeAllowed := FALSE;
ELSIF sv_NumberOfDevices[cCompEcoRobot] >= 1 THEN
   pbBool := GET_SYNC_REFTO("EcoRobot.sv_bUseEcoRobot", T#0s, s);
   IF pbBool^ THEN
      //eco robot switched on
      bScrapModeAllowed := FALSE;
   END_IF;
ELSIF sv_NumberOfDevices[cCompEuromap] >= 1 THEN
   pInterfaceType := GET_SYNC_REFTO("Euromap.sv_InterfaceType", T#0s, s);
   IF pInterfaceType^ <> nSwitchedOff THEN
      //euromap inerface switched on
      bScrapModeAllowed := FALSE;
   END_IF;
END_IF;

IF bScrapModeAllowed THEN
   FPlausSPCAction.iUpperLimit := 5;
ELSE
   FPlausSPCAction.iUpperLimit := 4;
END_IF;

;#END_EDIT_BLOCK END_FUNCTION

#END_OF_IEC_PART

@Puma @IecEditor 6 145 @Pou 25
@@@BEG_Comment@@@
@h    ! WARNING !
@h    The Kemro K2 system (including software) only meets category B according to EN 954-1,
@h    thus it is not intended for usage in safety-relevant control applications in the field
@h    of personal safety (e.g. emergency stop).
@h    To implement potentially necessary safety-relevant control tasks, always use additional
@h    external safety devices that are intended for the particular purpose, and meet the necessary
@h    functional safety.
@h    For further information see EN 954-1 (EN ISO 13849-1) and/or the K2-x00 user manual, chapter
@h    "CE conformity, directives and standards".

Plausibility function for SPC error / warn action
@@@END_Comment@@@

@BEG_Contents

@BEG_Func
@RT(17)FuncTreeContainer
1
@Var @RT(14)GET_SYNC_REFTO @RT(0) @T @T @DERIVED 0 @F @RT(34)KEBA_STANDARD_FUNCTION : ANY_REFTO @F
@T
@BEG_Attrib
0 @RT(0) @RT(0)
@END_Attrib
1 1 @F @F @F @F

@END_Func

@BEG_Const
@RT(18)ConstTreeContainer
1
@Var @RT(13)cCompEcoRobot @RT(0) @T @F @DT @RT(4)DINT @RT(0) @T @T @BASIC 0 @F
@F @F
@T
@BEG_Attrib
0 @RT(3)146 @RT(19)Component Eco Robot
@END_Attrib
1 1 @F @F @F @F

@END_Const

@BEG_Export

@BEG_Kind
@PLAUSIBILITY_FUNCTION @RT(15)FPlausSPCAction @STRUCTURED_TEXT
@RT(14)tsLimitDataINT @RT(0) @RT(0)
@END_Kind

@BEG_Dcl
@RT(16)DclTreeContainer
7
@Var @RT(11)DeviceClass @RT(0) @T @F @DT @RT(3)INT @RT(0) @T @T @BASIC 0 @F
@F @F
@T
@BEG_Attrib
3 @RT(0) @RT(0) @RT(0)
@END_Attrib
0 1 @F @F @F @F

@Var @RT(9)Userlevel @RT(0) @T @F @DT @RT(3)INT @RT(0) @T @T @BASIC 0 @F
@F @F
@T
@BEG_Attrib
3 @RT(0) @RT(0) @RT(0)
@END_Attrib
0 1 @F @F @F @F

@Var @RT(18)sv_NumberOfDevices @RT(0) @T @T @DERIVED 0 @T @T @DT @RT(17)tyNumberOfDevices @RT(0) @T @T @UNKNOWN 0 @F
@F @F
@T
@BEG_Attrib
3 @RT(0) @RT(0) @RT(0)
@END_Attrib
1 9 @F @F @F @F

@Var @RT(1)s @RT(0) @T @T @DERIVED 0 @F @RT(11)KSYS_Status @F
@T
@BEG_Attrib
3 @RT(0) @RT(0) @RT(0)
@END_Attrib
1 0 @F @F @F @F

@Var @RT(6)pbBool @RT(0) @T @T @REFTO 0 @T @DT @RT(4)BOOL @RT(0) @T @T @BASIC 0 @F
@F @F
@T
@BEG_Attrib
3 @RT(0) @RT(0) @RT(0)
@END_Attrib
1 0 @F @F @F @F

@Var @RT(14)pInterfaceType @RT(0) @T @T @REFTO 0 @F @DERIVED 0 @F @RT(16)tnRobotInterface @F
@T
@BEG_Attrib
3 @RT(0) @RT(0) @RT(0)
@END_Attrib
1 0 @F @F @F @F

@Var @RT(17)bScrapModeAllowed @RT(0) @T @F @DT @RT(4)BOOL @RT(0) @T @T @BASIC 0 @F
@F @F
@T
@BEG_Attrib
3 @RT(0) @RT(0) @RT(0)
@END_Attrib
1 0 @F @F @F @F

@END_Dcl

@END_Export

@BEG_Body
@TL(35)
(**************************************** WARNING ********************************************
 *** The KEBA Kemro K2 System including software is not intended for safety control tasks! ***
 ***                       For further information see Comment tab!                        ***
 *********************************************************************************************)

//"hold scrap" mode not allowed if Reject gate is available or
//robot switched on

FPlausSPCAction.iLowerLimit := 0;

bScrapModeAllowed := TRUE;
pbBool := GET_SYNC_REFTO("RejectGate1.do_RejectGate", T#0s, s);
IF s = KSYS_Status_OK THEN
   //reject gate available
   bScrapModeAllowed := FALSE;
ELSIF sv_NumberOfDevices[cCompEcoRobot] >= 1 THEN
   pbBool := GET_SYNC_REFTO("EcoRobot.sv_bUseEcoRobot", T#0s, s);
   IF pbBool^ THEN
      //eco robot switched on
      bScrapModeAllowed := FALSE;
   END_IF;
ELSIF sv_NumberOfDevices[cCompEuromap] >= 1 THEN
   pInterfaceType := GET_SYNC_REFTO("Euromap.sv_InterfaceType", T#0s, s);
   IF pInterfaceType^ <> nSwitchedOff THEN
      //euromap inerface switched on
      bScrapModeAllowed := FALSE;
   END_IF;
END_IF;

IF bScrapModeAllowed THEN
   FPlausSPCAction.iUpperLimit := 5;
ELSE
   FPlausSPCAction.iUpperLimit := 4;
END_IF;

@END_Body

@END_Contents
